FUNCTION_BLOCK TEMPLATE_FB
  {SET_ATTRIBUTE(OpcUa, SERVICE)}
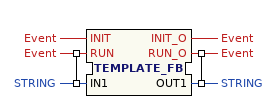
  EVENT_INPUT
    INIT;
    RUN WITH IN1;
  END_EVENT
  EVENT_OUTPUT
    INIT_O;
    RUN_O WITH OUT1;
  END_EVENT
  VAR_INPUT
    IN1 : STRING;
  END_VAR
  VAR_OUTPUT
    OUT1 : STRING;
  END_VAR
END_FUNCTION_BLOCK
